SUBAPPLICATION Uebung_209 (* Interlock: ILOCK_FB_RS (Zwei gegenseitig verriegelte Reset-Dominante Latches via AX2-Adapter) *)
  (* Standard: 61499-2; Description: Copyright (c) 2026 Meisterschulen am Ostbahnhof This program and the accompanying materials are made available under the terms of the Eclipse Public License 2.0 which is available at https://www.eclipse.org/legal/epl-2.0/ SPDX-License-Identifier: EPL-2.0 *)
  (* Version 1.0, 2026-05-07, Gemini CLI, Meisterschulen am Ostbahnhof, initial version using library block ILOCK_FB_RS *)
  PACKAGE Uebungen;
  IMPORT logiBUS::io::DI::logiBUS_DI::Input_I1;
  IMPORT logiBUS::io::DI::logiBUS_DI::Input_I2;
  IMPORT logiBUS::io::DI::logiBUS_DI::Input_I3;
  IMPORT logiBUS::io::DI::logiBUS_DI::Input_I4;
  IMPORT logiBUS::io::DQ::logiBUS_DO::Output_Q1;
  IMPORT logiBUS::io::DQ::logiBUS_DO::Output_Q2;
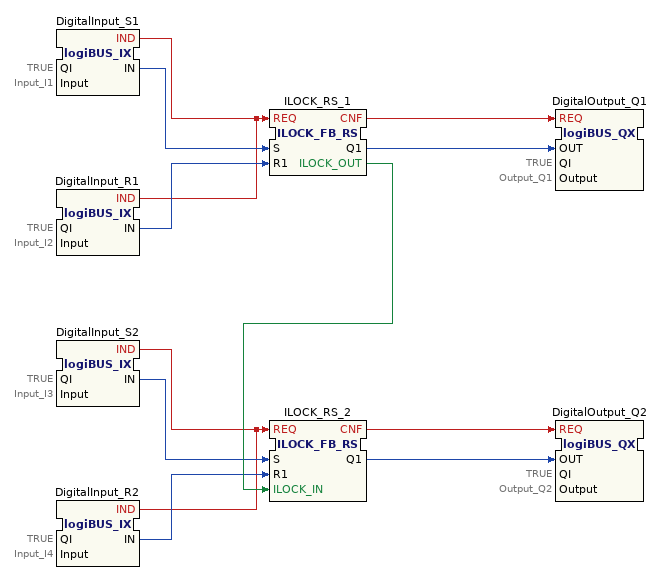
  FBS
    DigitalInput_S1 : logiBUS::io::DI::logiBUS_IX(QI := TRUE, Input := Input_I1);
    DigitalInput_R1 : logiBUS::io::DI::logiBUS_IX(QI := TRUE, Input := Input_I2);
    DigitalInput_S2 : logiBUS::io::DI::logiBUS_IX(QI := TRUE, Input := Input_I3);
    DigitalInput_R2 : logiBUS::io::DI::logiBUS_IX(QI := TRUE, Input := Input_I4);
    ILOCK_RS_1 : logiBUS::signalprocessing::interlock::ILOCK_FB_RS;
    ILOCK_RS_2 : logiBUS::signalprocessing::interlock::ILOCK_FB_RS;
    DigitalOutput_Q1 : logiBUS::io::DQ::logiBUS_QX(QI := TRUE, Output := Output_Q1);
    DigitalOutput_Q2 : logiBUS::io::DQ::logiBUS_QX(QI := TRUE, Output := Output_Q2);
  END_FBS
  EVENT_CONNECTIONS
    DigitalInput_S1.IND TO ILOCK_RS_1.REQ;
    DigitalInput_R1.IND TO ILOCK_RS_1.REQ;
    DigitalInput_S2.IND TO ILOCK_RS_2.REQ;
    DigitalInput_R2.IND TO ILOCK_RS_2.REQ;
    ILOCK_RS_1.CNF TO DigitalOutput_Q1.REQ;
    ILOCK_RS_2.CNF TO DigitalOutput_Q2.REQ;
  END_CONNECTIONS
  DATA_CONNECTIONS
    DigitalInput_S1.IN TO ILOCK_RS_1.S;
    DigitalInput_R1.IN TO ILOCK_RS_1.R1;
    DigitalInput_S2.IN TO ILOCK_RS_2.S;
    DigitalInput_R2.IN TO ILOCK_RS_2.R1;
    ILOCK_RS_1.Q1 TO DigitalOutput_Q1.OUT;
    ILOCK_RS_2.Q1 TO DigitalOutput_Q2.OUT;
  END_CONNECTIONS
  ADAPTER_CONNECTIONS
    ILOCK_RS_1.ILOCK_OUT TO ILOCK_RS_2.ILOCK_IN;
  END_CONNECTIONS
END_SUBAPPLICATION
